INTERFACE I_DatatypeVisitor

METHOD VisitDatatype
VAR_INPUT
	VisitingDatatype : I_Datatype;
END_VAR
END_METHOD

END_INTERFACE

(* stored: Version 1.1.0.1, ProductVersion 3.1.4024.12
   Itf I_DatatypeVisitor: Id {d84e842a-ff7a-036b-3d5a-ffd8731164fa}
   Method VisitDatatype: Id {187daa84-6e8c-0dee-2009-f0e41b495da3} *)
